TestInstancePath := AddTestNameToInstancePath(TestInstancePath := FindTestSuiteInstancePath());

AssertResults.ReportResult(ExpectedSize := SIZEOF(Expected),
                           ExpectedTypeClass := IBaseLibrary.TypeClass.TYPE_WSTRING,
                           ExpectedValue := ADR(Expected),
                           ActualSize := SIZEOF(Actual),
                           ActualTypeClass := IBaseLibrary.TypeClass.TYPE_WSTRING,
                           ActualValue := ADR(Actual),
                           Message := Message,
                           TestInstancePath := TestInstancePath,
                           AlreadyReported => AlreadyReported);

IF NOT AlreadyReported AND (Tc2_Standard.WLEN(STR := Expected) <> Tc2_Standard.WLEN(STR := Actual) OR (Expected <> Actual)) THEN
    SetTestFailed(AssertionType := E_AssertionType.Type_WSTRING,
                  AssertionMessage := Message);

    AssertMessageFormatter.LogAssertFailure(Expected := 'Not possible to print EXP unicode WSTRING value',
                                            Actual := 'Not possible to print ACT unicode WSTRING value',
                                            Message := Message,
                                            TestInstancePath := TestInstancePath);
END_IF
END_METHOD

(*
    Asserts that a condition is false. If it is not, an assertion error is created.
*)
METHOD PUBLIC AssertFalse
VAR_INPUT
    Condition : BOOL; // Condition to be checked
    Message : Tc2_System.T_MaxString; // The identifying message for the assertion error
END_VAR
AssertEquals_BOOL(Expected := FALSE, Actual := Condition, Message := Message);
END_METHOD

(*
    Asserts that a condition is true. If it is not, an assertion error is created.
*)
METHOD PUBLIC AssertTrue
VAR_INPUT
    Condition : BOOL; // Condition to be checked
    Message : Tc2_System.T_MaxString; // The identifying message for the assertion error
END_VAR
AssertEquals_BOOL(Expected := TRUE, Actual := Condition, Message := Message);
END_METHOD

METHOD INTERNAL CalculateAndSetNumberOfAssertsForTest
VAR_INPUT
    TestName : Tc2_System.T_MaxString;
END_VAR
VAR
    TestInstancePath : Tc2_System.T_MaxString;
    TotalNumberOfAsserts : UINT;
    NumberOfAsserts : UINT;
    NumberOfArrayAsserts : UINT;
    
    IteratorCounter : UINT;
END_VAR
TestInstancePath := AddTestNameToInstancePath(FindTestSuiteInstancePath());
NumberOfAsserts := AssertResults.GetNumberOfAssertsForTest(CompleteTestInstancePath := TestInstancePath);
NumberOfArrayAsserts := AssertArrayResults.GetNumberOfArrayAssertsForTest(CompleteTestInstancePath := TestInstancePath);
TotalNumberOfAsserts := NumberOfAsserts + NumberOfArrayAsserts;

IF TotalNumberOfAsserts > 0 THEN
    IF NumberOfTests > 0 THEN
        FOR IteratorCounter := 1 TO NumberOfTests BY 1 DO
            IF Tests[IteratorCounter].GetName() = TestName THEN
                Tests[IteratorCounter].SetNumberOfAssertions(NoOfAssertions := TotalNumberOfAsserts);
                RETURN;
            END_IF
        END_FOR
    END_IF
END_IF
END_METHOD

METHOD FB_init : BOOL
VAR_INPUT
    bInitRetains : BOOL; // if TRUE, the retain variables are initialized (warm start / cold start)
    bInCopyCode : BOOL;  // if TRUE, the instance afterwards gets moved into the copy code (online change)
END_VAR
GVL_TcUnit.NumberOfInitializedTestSuites := GVL_TcUnit.NumberOfInitializedTestSuites + 1;    
GVL_TcUnit.TestSuiteAddresses[GVL_TcUnit.NumberOfInitializedTestSuites] := THIS;
END_METHOD

(* Searches for the instance path of the calling function block *)
METHOD PRIVATE FindTestSuiteInstancePath : Tc2_System.T_MaxString
FindTestSuiteInstancePath := GetInstancePath();
END_METHOD

METHOD INTERNAL GetHasStartedRunning : BOOL
GetHasStartedRunning := HasStartedRunning;
END_METHOD

METHOD INTERNAL GetInstancePath : Tc2_System.T_MaxString
GetInstancePath := InstancePath;
END_METHOD

METHOD INTERNAL GetNumberOfFailedTests : UINT
VAR
    Counter : UINT;
    FailedTestsCount : UINT;
    NumberOfTestsToAnalyse : UINT(1..GVL_Param_TcUnit.MaxNumberOfTestSuites);
    NumberOfTestOverArrayLimit : UINT;
END_VAR
(* Limit the test analyse to the max array limit of 'Tests[]' *)
IF GetNumberOfTests() >  GVL_Param_TcUnit.MaxNumberOfTestsForEachTestSuite THEN
    NumberOfTestsToAnalyse := GVL_Param_TcUnit.MaxNumberOfTestsForEachTestSuite;
    NumberOfTestOverArrayLimit := GetNumberOfTests()-GVL_Param_TcUnit.MaxNumberOfTestsForEachTestSuite;
ELSE
    NumberOfTestsToAnalyse := GetNumberOfTests();
END_IF

IF NumberOfTests > 0 THEN
    FOR Counter := 1 TO NumberOfTestsToAnalyse BY 1 DO
        IF Tests[Counter].IsFailed() THEN
            FailedTestsCount := FailedTestsCount + 1;
        END_IF
    END_FOR
END_IF

GetNumberOfFailedTests := FailedTestsCount + NumberOfTestOverArrayLimit;
END_METHOD

METHOD INTERNAL GetNumberOfSkippedTests : UINT
VAR
    Counter : UINT;
    SkippedTestsCount : UINT;
    NumberOfTestsToAnalyse : UINT(1..GVL_Param_TcUnit.MaxNumberOfTestSuites);
END_VAR
(* Limit the test analyse to the max array limit of 'Tests[]' *)
IF GetNumberOfTests() >  GVL_Param_TcUnit.MaxNumberOfTestsForEachTestSuite THEN
    NumberOfTestsToAnalyse := GVL_Param_TcUnit.MaxNumberOfTestsForEachTestSuite;
ELSE
    NumberOfTestsToAnalyse := GetNumberOfTests();
END_IF

IF NumberOfTests > 0 THEN
    FOR Counter := 1 TO NumberOfTestsToAnalyse BY 1 DO
        IF Tests[Counter].IsSkipped() THEN
            SkippedTestsCount := SkippedTestsCount + 1;
        END_IF
    END_FOR
END_IF

GetNumberOfSkippedTests := SkippedTestsCount;
END_METHOD

METHOD INTERNAL GetNumberOfSuccessfulTests : UINT
GetNumberOfSuccessfulTests := GetNumberOfTests() - GetNumberOfFailedTests() - GetNumberOfSkippedTests();
END_METHOD

METHOD INTERNAL GetNumberOfTests : UINT
GetNumberOfTests := NumberOfTests;
END_METHOD

(* This method returns the test at the n'th position, ranging from 1.. NumberOfTests *)
METHOD INTERNAL GetTestByPosition : FB_Test
VAR_INPUT
    Position : UINT(1..GVL_Param_TcUnit.MaxNumberOfTestsForEachTestSuite);
END_VAR
GetTestByPosition := Tests[Position];
END_METHOD

METHOD INTERNAL GetTestOrderNumber : UINT(0..GVL_Param_TcUnit.MaxNumberOfTestsForEachTestSuite);
VAR_INPUT
    TestName : Tc2_System.T_MaxString;
END_VAR
VAR
    IteratorCounter : UINT;
    NumberOfTestsToAnalyse : UINT(1..GVL_Param_TcUnit.MaxNumberOfTestSuites);
END_VAR
(* Limit the test analyse to the max array limit of 'Tests[]' *)
IF NumberOfTests >  GVL_Param_TcUnit.MaxNumberOfTestsForEachTestSuite THEN
    NumberOfTestsToAnalyse := GVL_Param_TcUnit.MaxNumberOfTestsForEachTestSuite;
ELSE
    NumberOfTestsToAnalyse := NumberOfTests;
END_IF

IF NumberOfTests > 0 THEN
    FOR IteratorCounter := 1 TO NumberOfTestsToAnalyse BY 1 DO
        IF Tests[IteratorCounter].GetName() = TestName THEN
            GetTestOrderNumber := Tests[IteratorCounter].GetTestOrder();
            RETURN;
        END_IF
    END_FOR
END_IF
END_METHOD

METHOD INTERNAL IsTestFinished : BOOL
VAR_INPUT
    TestName : Tc2_System.T_MaxString;
END_VAR
VAR
    IteratorCounter : UINT;
    NumberOfTestsToAnalyse : UINT(0..GVL_Param_TcUnit.MaxNumberOfTestsForEachTestSuite);
END_VAR
(* Limit the test analyse to the max array limit of 'Tests[]' *)
IF NumberOfTests >  GVL_Param_TcUnit.MaxNumberOfTestsForEachTestSuite THEN
    NumberOfTestsToAnalyse := GVL_Param_TcUnit.MaxNumberOfTestsForEachTestSuite;
ELSE
    NumberOfTestsToAnalyse := NumberOfTests;
END_IF

IsTestFinished := FALSE;
IF NumberOfTests > 0 THEN
    FOR IteratorCounter := 1 TO NumberOfTestsToAnalyse BY 1 DO
        IF Tests[IteratorCounter].GetName() = TestName THEN
            IsTestFinished := Tests[IteratorCounter].IsFinished();
            RETURN;
        END_IF
    END_FOR
END_IF
END_METHOD

METHOD INTERNAL SetHasStartedRunning
HasStartedRunning := TRUE;
END_METHOD

METHOD PRIVATE SetTestFailed
VAR_INPUT
    AssertionType : E_AssertionType;
    AssertionMessage : Tc2_System.T_MaxString;
END_VAR
VAR
    IteratorCounter : UINT;
    NumberOfTestsToAnalyse : UINT(0..GVL_Param_TcUnit.MaxNumberOfTestsForEachTestSuite);
END_VAR
(* Limit the test analyse to the max array limit of 'Tests[]' *)
IF NumberOfTests >  GVL_Param_TcUnit.MaxNumberOfTestsForEachTestSuite THEN
    NumberOfTestsToAnalyse := GVL_Param_TcUnit.MaxNumberOfTestsForEachTestSuite;
ELSE
    NumberOfTestsToAnalyse := NumberOfTests;
END_IF

IF NumberOfTests > 0 THEN
    FOR IteratorCounter := 1 TO NumberOfTestsToAnalyse BY 1 DO
        IF Tests[IteratorCounter].GetName() = GVL_TcUnit.CurrentTestNameBeingCalled THEN
            Tests[IteratorCounter].SetFailed();
            Tests[IteratorCounter].SetAssertionType(AssertType := AssertionType);
            Tests[IteratorCounter].SetAssertionMessage(AssertMessage := AssertionMessage);
        END_IF
    END_FOR
END_IF
END_METHOD

(* Marks the test as finished in this testsuite.
   Returns TRUE if test was found, and FALSE if a test with this name was not found in this testsuite
*)
METHOD INTERNAL SetTestFinished : BOOL;
VAR_INPUT
    TestName : Tc2_System.T_MaxString;
END_VAR
VAR
    IteratorCounter : UINT;
    NumberOfTestsToAnalyse : UINT(0..GVL_Param_TcUnit.MaxNumberOfTestsForEachTestSuite);
END_VAR
(* Limit the test analyse to the max array limit of 'Tests[]' *)
IF NumberOfTests >  GVL_Param_TcUnit.MaxNumberOfTestsForEachTestSuite THEN
    NumberOfTestsToAnalyse := GVL_Param_TcUnit.MaxNumberOfTestsForEachTestSuite;
ELSE
    NumberOfTestsToAnalyse := NumberOfTests;
END_IF
IF NumberOfTests > 0 THEN
    FOR IteratorCounter := 1 TO NumberOfTestsToAnalyse BY 1 DO
        IF Tests[IteratorCounter].GetName() = TestName THEN
            Tests[IteratorCounter].SetFinished();
            SetTestFinished := TRUE;
            RETURN;
        END_IF
    SetTestFinished := FALSE;
    END_FOR
END_IF
END_METHOD

END_FUNCTION_BLOCK

// POUs/FB_xUnitXmlPublisher
(*
    Publishes test results into an xUnit compatible Xml file
*)
FUNCTION_BLOCK FB_xUnitXmlPublisher IMPLEMENTS I_TestResultLogger
VAR
    // Dependancy Injection via FB_Init
    TestResults : I_TestResults;

    // File access mode
    AccessMode : SysFile.ACCESS_MODE := SysFile.AM_WRITE_PLUS;

    File : FB_FileControl;
    Xml : FB_XMLControl;
    BufferInitialised : BOOL := FALSE;
    Buffer : ARRAY [0..(GVL_Param_TcUnit.XUnitBufferSize - 1)] OF BYTE;
    WritingTestSuiteResultNumber : UINT(1..GVL_Param_TcUnit.MaxNumberOfTestSuites);
    PublishTrigger : Tc2_Standard.R_TRIG;
END_VAR

(*
    Deletes the former file (if it exists).
    Opens the file, writes the buffer and closes it.
*)
METHOD PRIVATE DeleteOpenWriteClose : SysFile.SysTypes.RTS_IEC_RESULT;
DeleteOpenWriteClose := SysDir.CmpErrors.Errors.ERR_OK;   
IF Initialised() THEN
    DeleteOpenWriteClose := MAX(DeleteOpenWriteClose, File.Delete(Filename := GVL_Param_TcUnit.xUnitFilePath));
    DeleteOpenWriteClose := MAX(DeleteOpenWriteClose, File.Open(Filename := GVL_Param_TcUnit.xUnitFilePath, FileAccessMode := AccessMode));
    DeleteOpenWriteClose := MAX(DeleteOpenWriteClose, File.Write(BufferPointer := ADR(Buffer), Xml.Length)); 
    DeleteOpenWriteClose := MAX(DeleteOpenWriteClose, File.Close());
ELSE
    DeleteOpenWriteClose := SysDir.CmpErrors.Errors.ERR_NOBUFFER;
END_IF;
END_METHOD

(*
    FB_Init is always available implicitly AND it is used primarily FOR initialization.
    The return value is not evaluated. For a specific influence, you can also declare the
    methods explicitly and provide additional code there with the standard initialization
    code. You can evaluate the return value.
*)
METHOD FB_Init: BOOL
VAR_INPUT
    bInitRetains: BOOL; // TRUE: the retain variables are initialized (reset warm / reset cold)
    bInCopyCode: BOOL;  // TRUE: the instance will be copied to the copy code afterward (online change)
    iTestResults : I_TestResults; // Interface dependency injection
END_VAR
// Set buffer and flag
Xml.SetBuffer(PointerToBuffer := ADR(Buffer), SizeOfBuffer := SIZEOF(Buffer));

// Set buffer initialised
BufferInitialised := TRUE;

// Set testresult interface
TestResults := iTestResults;
END_METHOD

METHOD PRIVATE Initialised : BOOL
Initialised := THIS^.BufferInitialised;
END_METHOD

(*
    This method is responsible for the entire generation of the output file. 
    The output of the xml writer is NOT beautified.
    
    When new data is available, feel free to add it to the report
*)
METHOD PUBLIC LogTestSuiteResults
VAR
    UnitTestResults : REFERENCE TO ST_TestSuiteResults;
    CurrentSuiteNumber : UINT;
    CurrentTestCount : UINT;
END_VAR
VAR CONSTANT
    TEST_STATUS_SKIP : STRING := 'SKIP';
    TEST_STATUS_PASS : STRING := 'PASS';
    TEST_STATUS_FAIL : STRING := 'FAIL';
END_VAR
UnitTestResults REF=TestResults.GetTestSuiteResults();

// Only publish once if "GVL_Param_TcUnit.xUnitEnablePublish" is enabled and all test results are stored.
PublishTrigger(CLK := (TestResults.GetAreTestResultsAvailable() AND GVL_Param_TcUnit.xUnitEnablePublish));
IF PublishTrigger.Q THEN

    (* <?xml version="1.0" encoding="UTF-8"?> *)
    Xml.WriteDocumentHeader(Header := '<?xml version="1.0" encoding="UTF-8"?>');

    (* <testsuites> *)
    Xml.NewTag('testsuites');
    Xml.NewParameter('disabled', '');
    Xml.NewParameter('failures', UINT_TO_STRING(UnitTestResults.NumberOfFailedTestCases));
    Xml.NewParameter('tests', UINT_TO_STRING(UnitTestResults.NumberOfSuccessfulTestCases));

    FOR CurrentSuiteNumber := 1 TO UnitTestResults.NumberOfTestSuites BY 1 DO 
        (* <testsuite> *)
        Xml.NewTag('testsuite');
        Xml.NewParameter('id', UINT_TO_STRING(UnitTestResults.TestSuiteResults[CurrentSuiteNumber].Identity));
        Xml.NewParameter('name', UnitTestResults.TestSuiteResults[CurrentSuiteNumber].name);
        Xml.NewParameter('tests', UINT_TO_STRING(UnitTestResults.TestSuiteResults[CurrentSuiteNumber].NumberOfTests));        
        Xml.NewParameter('failures', UINT_TO_STRING(UnitTestResults.TestSuiteResults[CurrentSuiteNumber].NumberOfFailedTests));

        FOR CurrentTestCount := 1 TO UnitTestResults.TestSuiteResults[CurrentSuiteNumber].NumberOfTests BY 1 DO
            (* <testcase> *)
            Xml.NewTag('testcase');
            Xml.NewParameter('name', UnitTestResults.TestSuiteResults[CurrentSuiteNumber].TestCaseResults[CurrentTestCount].TestName);
            Xml.NewParameter('classname', UnitTestResults.TestSuiteResults[CurrentSuiteNumber].TestCaseResults[CurrentTestCount].TestClassName);

            IF UnitTestResults.TestSuiteResults[CurrentSuiteNumber].TestCaseResults[CurrentTestCount].TestIsFailed THEN
                Xml.NewParameter('status', TEST_STATUS_FAIL);
            ELSIF UnitTestResults.TestSuiteResults[CurrentSuiteNumber].TestCaseResults[CurrentTestCount].TestIsSkipped THEN   
                Xml.NewParameter('status', TEST_STATUS_SKIP);
            ELSE
                Xml.NewParameter('status', TEST_STATUS_PASS);
            END_IF

            (* Determine testcase fail or success *)
            IF UnitTestResults.TestSuiteResults[CurrentSuiteNumber].TestCaseResults[CurrentTestCount].FailureType <> E_AssertionType.Type_UNDEFINED THEN 
                (* In case of fail 
                    <failure message="Values differ" type="BYTE" />
                *)
                Xml.NewTag('failure');
                Xml.NewParameter('message', UnitTestResults.TestSuiteResults[CurrentSuiteNumber].TestCaseResults[CurrentTestCount].FailureMessage);
                Xml.NewParameter('type', F_AssertionTypeToString(UnitTestResults.TestSuiteResults[CurrentSuiteNumber].TestCaseResults[CurrentTestCount].FailureType));       
                (* Close failure tag *)
                Xml.CloseTag();
            ELSE
            (* In case of success *)
            Xml.NewTagData('');

            END_IF
            (* Close testcase tag*)         
            Xml.CloseTag();

        END_FOR
        (* Close testsuite tag *)
        Xml.CloseTag();

    END_FOR
    (* Close testsuites *)
    Xml.CloseTag();

    (* Delete, open, save and close the file *)
    DeleteOpenWriteClose();

    (* Clear the internal buffer *)
    Xml.ClearBuffer();

    (* Inform user *)
    GVL_TcUnit.AdsMessageQueue.WriteLog(MsgCtrlMask := Tc2_System.ADSLOG_MSGTYPE_HINT,
                                        msgFmtStr := '%s',
                                        strArg := '| ==========TEST RESULTS EXPORTED===========');
                                                                                         
    GVL_TcUnit.AdsMessageQueue.WriteLog(MsgCtrlMask := Tc2_System.ADSLOG_MSGTYPE_HINT,   
                                        msgFmtStr :=  '| Location: %s ',                 
                                        strArg := GVL_Param_TcUnit.xUnitFilePath);            

    GVL_TcUnit.AdsMessageQueue.WriteLog(MsgCtrlMask := Tc2_System.ADSLOG_MSGTYPE_HINT,
                                        MsgFmtStr := '%s',                               
                                        StrArg := '| ======================================');
END_IF
END_METHOD

END_FUNCTION_BLOCK
